TYPE TFMachinePalletizer_Pallet_OLD :
STRUCT
	X			: REAL	:= 0.0;	(* READ	- (mm) Dimensione X *)
	Y			: REAL	:= 0.0;	(* READ	- (mm) Dimensione Y *)
	Z			: REAL	:= 0.0;	(* READ	- (mm) Dimensione Z *)
END_STRUCT
END_TYPE

(* stored: Version 1.1.0.1, ProductVersion 3.1.4024.11
   DUT TFMachinePalletizer_Pallet_OLD: Id {c8fa156f-6512-41ac-bea1-82aaa0dc6adf} *)
